TYPE T_Ctrl_SIf_GRN_Cfg :
STRUCT
END_STRUCT
END_TYPE

(* stored: Version 1.1.0.1, ProductVersion 3.1.0.25
   DUT T_Ctrl_SIf_GRN_Cfg: Id {4330c1f4-231e-43ce-bcf1-0e60f4afa87b} *)
